Fanuc KAREL source: kt00602.KL

-- PROVISIONAL review KL for V770-1; original PC SHA256 2f3ef2cd7cd4e6da5fa7d9378e9af6c8b226132c2d7608fed3ad6b46f7cdc961
-- Incomplete behavior may be omitted. Consult companion uncertainty JSON. Do not deploy.
PROGRAM KT00602
%NOLOCKGROUP
VAR
  I1 : INTEGER
  I2 : INTEGER
  OUT : REAL
BEGIN
  -- UNRESOLVED_PC offsets 5-16; opcodes 2E,23
  -- UNRESOLVED_PC offsets 21-32; opcodes 2E,23
  -- UNRESOLVED_PC offsets 37-48; opcodes 2E,23
  -- UNRESOLVED_PC offsets 53-64; opcodes 2E,23
  -- UNRESOLVED_PC offsets 69-82; opcodes 21,64,23
  -- UNRESOLVED_PC offsets 87-91; opcodes 7F
END KT00602
